(* IEC 61131-3 sources: IEC61131-3-CDSV3/Regular Expressions/src/20 Program Organization Units, 8 files *)

(* ---- FuCompiledPatternAnsiToW.pou ---- *)
(*#-#-#-#-#-#-#-#-#-#---Declaration---#-#-#-#-#-#-#-#-#-#-#-#-#*)

// Converts an ANSI/ISO 8859-1 compiled pattern to an Unicode compiled pattern.
// ANSI/ISO 8859-1 compiled patterns can be converted to Unicode without any loss.
FUNCTION FuCompiledPatternAnsiToW : typCompiledPatternW
VAR_INPUT
    typPattern: typCompiledPattern;
END_VAR
{library PRIVATE}
VAR
    i: UDINT;
END_VAR
(*#-#-#-#-#-#-#-#-#-#---Implementation---#-#-#-#-#-#-#-#-#-#-#-#-#*)

IF typPattern.uiCountTokens = 0 THEN
    RETURN;
END_IF

FuCompiledPatternAnsiToW.xCaseInsensitive := typPattern.xCaseInsensitive;
FuCompiledPatternAnsiToW.uiCountTokens := typPattern.uiCountTokens;

FOR i := 0 TO TO_UDINT((typPattern.uiCountTokens - 1)) BY 1 DO
    FuCompiledPatternAnsiToW.atTokens[i].eType := typPattern.atTokens[i].eType;
    FuCompiledPatternAnsiToW.atTokens[i].dwChar := TO_DWORD(typPattern.atTokens[i].bChar);
    FuCompiledPatternAnsiToW.atTokens[i].dwAlternativeChar := TO_DWORD(typPattern.atTokens[i].bAlternativeChar);
END_FOR

(* ---- FuCompilePattern.pou ---- *)
(*#-#-#-#-#-#-#-#-#-#---Declaration---#-#-#-#-#-#-#-#-#-#-#-#-#*)

// Compiles the pattern into a stream of tokens for matching.
// The ISO 8859-1 latin alphabet can be matched case insensitive,
// otherwise by default the pattern is case sensitive.
//
// A few examples of valid patterns:
//  - 'A*bEd'
//  - 'A*?bEd'
//  - 'A.b*e*'
//  - '*A\.b\*e*'
//  - 'A?\bed'
//
// The return value signifies whether compilation was successful,
// or the given pattern is invalid.
{attribute 'qualified_only'}
FUNCTION FuCompilePattern : BOOL
VAR_INPUT
    sPattern: STRING(255);              // The pattern string to compile
    xCaseInsensitive: BOOL := FALSE;    // Whether the pattern is case insensitive (ISO 8859-1 latin1)
END_VAR
VAR_OUTPUT
    typPattern: typCompiledPattern;     // The compiled pattern, for "FuMatchExpression"
END_VAR
{library PRIVATE}
VAR
    i: UINT;

    tempChar: BYTE;
    tempNextChar: BYTE;
    tempIndex: UINT;

    tempMaxStrIndex: UINT;
END_VAR
VAR CONSTANT
    CHAR_WILDCARD: BYTE := 42; // *
    CHAR_LAZINESS: BYTE := 63; // ?
    CHAR_DOT: BYTE := 46; // .
    CHAR_ESCAPE: BYTE := 92; // \
END_VAR
(*#-#-#-#-#-#-#-#-#-#---Implementation---#-#-#-#-#-#-#-#-#-#-#-#-#*)

FuCompilePattern := FALSE;

IF sPattern = '' THEN
    RETURN;
END_IF

tempMaxStrIndex := TO_UINT(Standard.LEN(sPattern)) - 1;

FOR i := 0 TO tempMaxStrIndex BY 1 DO
    IF sPattern[i] = 0 OR_ELSE tempIndex > ParameterList.uiMaxPatternTokens THEN
        EXIT;
    END_IF

    tempChar := TO_BYTE(sPattern[i]);

    IF i < tempMaxStrIndex THEN
        tempNextChar := TO_BYTE(sPattern[(i + 1)]);
    ELSE
        tempNextChar := 0;
    END_IF

    IF tempChar = CHAR_WILDCARD THEN // Wildcard (*)
        typPattern.atTokens[tempIndex].eType := eTokenType.WILDCARD;
        typPattern.atTokens[tempIndex].bChar := 0; // Use bChar as modifier to be lazy
    ELSIF
        tempChar = CHAR_LAZINESS AND_THEN
        tempIndex > 0 AND_THEN
        typPattern.atTokens[(tempIndex - 1)].eType = eTokenType.WILDCARD
    THEN // Laziness (?), but only if previously wildcard, otherwise literal
        typPattern.atTokens[(tempIndex - 1)].bChar := 1;
        CONTINUE;
    ELSIF tempChar = CHAR_DOT THEN // Single char (.)
        typPattern.atTokens[tempIndex].eType := eTokenType.ANYCHAR;
    ELSIF
        tempChar = CHAR_ESCAPE AND_THEN (
            tempNextChar = CHAR_WILDCARD OR_ELSE
            tempNextChar = CHAR_DOT
        )
    THEN // Backslash (escape token for . or *, if followed by . or *)
        typPattern.atTokens[tempIndex].eType := eTokenType.LITERAL;
        typPattern.atTokens[tempIndex].bChar := tempNextChar;
        i := i + 1;
    ELSE
        typPattern.atTokens[tempIndex].eType := eTokenType.LITERAL;
        typPattern.atTokens[tempIndex].bChar := tempChar;

        tempNextChar := 0;
        IF xCaseInsensitive THEN
            // Calculate for the ISO 8859-1 latin1 alphabet the uppercase or lowercase character number
            IF tempChar >= 65 AND_THEN tempChar <= 90 THEN
                // Uppercase A-Z
                tempNextChar := tempChar + 32;
            ELSIF tempChar >= 97 AND_THEN tempChar <= 122 THEN
                // Lowercase a-z
                tempNextChar := tempChar - 32;
            ELSIF tempChar >= 192 AND_THEN tempChar <= 221 AND_THEN tempChar <> 215 THEN
                // Uppercase ISO 8859-1
                tempNextChar := tempChar + 32;
            ELSIF tempChar >= 224 AND_THEN tempChar <= 253 AND_THEN tempChar <> 247 THEN
                // Lowercase ISO 8859-1
                tempNextChar := tempChar - 32;
            END_IF
        END_IF

        typPattern.atTokens[tempIndex].bAlternativeChar := tempNextChar;
    END_IF

    tempIndex := tempIndex + 1;
    typPattern.uiCountTokens := tempIndex;
END_FOR

FuCompilePattern := (tempIndex > 0);
typPattern.xCaseInsensitive := xCaseInsensitive;

(* ---- FuCompilePatternUTF8.pou ---- *)
(*#-#-#-#-#-#-#-#-#-#---Declaration---#-#-#-#-#-#-#-#-#-#-#-#-#*)

// Compiles the pattern into a stream of tokens for matching.
// This is the UTF-8 version of FuCompilePattern.
//
// Disabling strict conformity allows the usage of the extended ASCII alphabet (ISO 8859-1, decimal 160-255),
// as long as it doesn't form a valid UTF-8 byte sequence.
//
// The alphabet can be matched case insensitive,
// otherwise by default the pattern is case sensitive.
// The case mapping table is NOT completely covered,
// as such you MAY encounter missing case conversion
// for some languages.
//
// A few examples of valid patterns:
//  - 'A*bEd'
//  - 'A*?bEd'
//  - 'A.b*e*'
//  - '*A\.b\*e*'
//  - 'A?\bed'
//
// The return value signifies whether compilation was successful,
// or the given pattern is invalid.
{attribute 'qualified_only'}
FUNCTION FuCompilePatternUTF8 : BOOL
VAR_INPUT
    psPattern: POINTER TO STRING(1);      // The pattern string to compile - for technical reasons this is a STRING(1), although any length is supported
    udiPatternLength: UDINT;              // Pattern string length (in bytes, not codepoints)
    xCaseInsensitive: BOOL := FALSE;      // Whether the pattern is case insensitive
    xStrictConformity: BOOL := TRUE;      // Require strict conformity to the Unicode standard
END_VAR
VAR_OUTPUT
    typPattern: typCompiledPatternW;      // The compiled pattern, for "FuMatchExpressionUTF8"
END_VAR
{library PRIVATE}
VAR
    tempPointer: POINTER TO STRING(1);

    i: UDINT;

    tempChar: DWORD;
    tempCharLength: UDINT;

    tempNextChar: DWORD;
    tempNextCharLength: UDINT;

    tempIndex: UINT;
    tempMaxStrIndex: UDINT;
END_VAR
VAR CONSTANT
    CHAR_WILDCARD: DWORD := 42; // *
    CHAR_LAZINESS: DWORD := 63; // ?
    CHAR_DOT: DWORD := 46; // .
    CHAR_ESCAPE: DWORD := 92; // \
END_VAR
(*#-#-#-#-#-#-#-#-#-#---Implementation---#-#-#-#-#-#-#-#-#-#-#-#-#*)

FuCompilePatternUTF8 := FALSE;

IF udiPatternLength = 0 THEN
    RETURN;
END_IF

tempPointer := psPattern;

i := 0;
tempMaxStrIndex := udiPatternLength - 1;

WHILE i <= tempMaxStrIndex DO
    IF tempIndex > ParameterList.uiMaxPatternTokens THEN
        EXIT;
    END_IF

    IF
        NOT FuUtf8CharToDword(
            psInput := (tempPointer + i),
            udiStringLength := (udiPatternLength - i),
            xStrictConformity := xStrictConformity,
            dwCodepoint => tempChar,
            usiByteLength => tempCharLength
        )
    THEN
        RETURN;
    END_IF

    IF tempChar = 0 THEN
        EXIT;
    END_IF

    IF
        i > tempMaxStrIndex OR_ELSE
        NOT FuUtf8CharToDword(
            psInput := (tempPointer + i + tempCharLength),
            udiStringLength := (udiPatternLength - i),
            xStrictConformity := xStrictConformity,
            dwCodepoint => tempNextChar,
            usiByteLength => tempNextCharLength
        )
    THEN
        tempNextChar := 0;
        tempNextCharLength := 0;
    END_IF

    IF tempChar = CHAR_WILDCARD THEN // Wildcard (*)
        typPattern.atTokens[tempIndex].eType := eTokenType.WILDCARD;
        typPattern.atTokens[tempIndex].dwChar := 0; // Use dwChar as modifier to be lazy
    ELSIF
        tempChar = CHAR_LAZINESS AND_THEN
        tempIndex > 0 AND_THEN
        typPattern.atTokens[(tempIndex - 1)].eType = eTokenType.WILDCARD
    THEN // Laziness (?), but only if previously wildcard, otherwise literal
        typPattern.atTokens[(tempIndex - 1)].dwChar := 1;

        i := i + tempCharLength;
        CONTINUE;
    ELSIF tempChar = CHAR_DOT THEN // Single char (.)
        typPattern.atTokens[tempIndex].eType := eTokenType.ANYCHAR;
    ELSIF
        tempChar = CHAR_ESCAPE AND_THEN (
            tempNextChar = CHAR_WILDCARD OR_ELSE
            tempNextChar = CHAR_DOT
        )
    THEN // Backslash (escape token for . or *, if followed by . or *)
        typPattern.atTokens[tempIndex].eType := eTokenType.LITERAL;
        typPattern.atTokens[tempIndex].dwChar := tempNextChar;
        i := i + tempNextCharLength;
    ELSE
        typPattern.atTokens[tempIndex].eType := eTokenType.LITERAL;
        typPattern.atTokens[tempIndex].dwChar := tempChar;

        IF xCaseInsensitive THEN
            // Calculate for the ISO 8859-1 latin1 alphabet the uppercase or lowercase character number (efficient way)
            IF tempChar >= 65 AND_THEN tempChar <= 90 THEN
                // Uppercase A-Z
                tempNextChar := tempChar + 32;
            ELSIF tempChar >= 97 AND_THEN tempChar <= 122 THEN
                // Lowercase a-z
                tempNextChar := tempChar - 32;
            ELSIF tempChar >= 192 AND_THEN tempChar <= 221 AND_THEN tempChar <> 215 THEN
                // Uppercase ISO 8859-1
                tempNextChar := tempChar + 32;
            ELSIF tempChar >= 224 AND_THEN tempChar <= 253 AND_THEN tempChar <> 247 THEN
                // Lowercase ISO 8859-1
                tempNextChar := tempChar - 32;
            ELSE
                // If we're not in the ISO 8859-1 latin1 alphabet range, use the Unicode function to calculate it
                tempNextChar := FuUnicodeCodepointCaseConvert(tempChar);
            END_IF
        ELSE
            tempNextChar := 0;
        END_IF

        typPattern.atTokens[tempIndex].dwAlternativeChar := tempNextChar;
    END_IF

    tempIndex := tempIndex + 1;
    typPattern.uiCountTokens := tempIndex;

    i := i + tempCharLength;
END_WHILE

FuCompilePatternUTF8 := (tempIndex > 0);
typPattern.xCaseInsensitive := xCaseInsensitive;

(* ---- FuCompilePatternW.pou ---- *)
(*#-#-#-#-#-#-#-#-#-#---Declaration---#-#-#-#-#-#-#-#-#-#-#-#-#*)

// Compiles the pattern into a stream of tokens for matching.
// This is the UTF-16 (WSTRING) version of FuCompilePattern.
//
// The alphabet can be matched case insensitive,
// otherwise by default the pattern is case sensitive.
// The case mapping table is NOT completely covered,
// as such you MAY encounter missing case conversion
// for some languages.
//
// A few examples of valid patterns:
//  - 'A*bEd'
//  - 'A*?bEd'
//  - 'A.b*e*'
//  - '*A\.b\*e*'
//  - 'A?\bed'
//
// The return value signifies whether compilation was successful,
// or the given pattern is invalid.
{attribute 'qualified_only'}
FUNCTION FuCompilePatternW : BOOL
VAR_INPUT
    pwsPattern: POINTER TO WSTRING(1);    // The pattern string to compile - for technical reasons this is a WSTRING(1), although any length is supported
    udiPatternLength: UDINT;              // Pattern string length (in words (length in bytes/2), not codepoints)
    xCaseInsensitive: BOOL := FALSE;      // Whether the pattern is case insensitive
END_VAR
VAR_OUTPUT
    typPattern: typCompiledPatternW;      // The compiled pattern, for "FuMatchExpressionW"
END_VAR
{library PRIVATE}
VAR
    tempPointer: POINTER TO WSTRING(1);

    i: UDINT;

    tempChar: DWORD;
    tempCharLength: UDINT;

    tempNextChar: DWORD;
    tempNextCharLength: UDINT;

    tempIndex: UINT;
    tempMaxStrIndex: UDINT;
END_VAR
VAR CONSTANT
    CHAR_WILDCARD: DWORD := 42; // *
    CHAR_LAZINESS: DWORD := 63; // ?
    CHAR_DOT: DWORD := 46; // .
    CHAR_ESCAPE: DWORD := 92; // \
END_VAR
(*#-#-#-#-#-#-#-#-#-#---Implementation---#-#-#-#-#-#-#-#-#-#-#-#-#*)

FuCompilePatternW := FALSE;

IF udiPatternLength = 0 THEN
    RETURN;
END_IF

tempPointer := pwsPattern;

i := 0;
tempMaxStrIndex := udiPatternLength - 1;

WHILE i <= tempMaxStrIndex DO
    IF tempIndex > ParameterList.uiMaxPatternTokens THEN
        EXIT;
    END_IF

    IF NOT FuUtf16CharToDword(psInput := (tempPointer + (i * 2)), udiStringLength := (udiPatternLength - (i * 2)), dwCodepoint => tempChar, usiWordLength => tempCharLength) THEN
        RETURN;
    END_IF

    IF tempChar = 0 THEN
        EXIT;
    END_IF

    IF
        i > tempMaxStrIndex OR_ELSE
        NOT FuUtf16CharToDword(
            psInput := (tempPointer + (i * 2) + (tempCharLength * 2)),
            udiStringLength := (udiPatternLength - (i * 2) - (tempCharLength * 2)),
            dwCodepoint => tempNextChar,
            usiWordLength => tempNextCharLength
        )
    THEN
        tempNextChar := 0;
        tempNextCharLength := 0;
    END_IF

    IF tempChar = CHAR_WILDCARD THEN // Wildcard (*)
        typPattern.atTokens[tempIndex].eType := eTokenType.WILDCARD;
        typPattern.atTokens[tempIndex].dwChar := 0; // Use dwChar as modifier to be lazy
    ELSIF
        tempChar = CHAR_LAZINESS AND_THEN
        tempIndex > 0 AND_THEN
        typPattern.atTokens[(tempIndex - 1)].eType = eTokenType.WILDCARD
    THEN // Laziness (?), but only if previously wildcard, otherwise literal
        typPattern.atTokens[(tempIndex - 1)].dwChar := 1;

        i := i + tempCharLength;
        CONTINUE;
    ELSIF tempChar = CHAR_DOT THEN // Single char (.)
        typPattern.atTokens[tempIndex].eType := eTokenType.ANYCHAR;
    ELSIF
        tempChar = CHAR_ESCAPE AND_THEN (
            tempNextChar = CHAR_WILDCARD OR_ELSE
            tempNextChar = CHAR_DOT
        )
    THEN // Backslash (escape token for . or *, if followed by . or *)
        typPattern.atTokens[tempIndex].eType := eTokenType.LITERAL;
        typPattern.atTokens[tempIndex].dwChar := tempNextChar;
        i := i + tempNextCharLength;
    ELSE
        typPattern.atTokens[tempIndex].eType := eTokenType.LITERAL;
        typPattern.atTokens[tempIndex].dwChar := tempChar;

        IF xCaseInsensitive THEN
            // Calculate for the ISO 8859-1 latin1 alphabet the uppercase or lowercase character number (efficient way)
            IF tempChar >= 65 AND_THEN tempChar <= 90 THEN
                // Uppercase A-Z
                tempNextChar := tempChar + 32;
            ELSIF tempChar >= 97 AND_THEN tempChar <= 122 THEN
                // Lowercase a-z
                tempNextChar := tempChar - 32;
            ELSIF tempChar >= 192 AND_THEN tempChar <= 221 AND_THEN tempChar <> 215 THEN
                // Uppercase ISO 8859-1
                tempNextChar := tempChar + 32;
            ELSIF tempChar >= 224 AND_THEN tempChar <= 253 AND_THEN tempChar <> 247 THEN
                // Lowercase ISO 8859-1
                tempNextChar := tempChar - 32;
            ELSE
                // If we're not in the ISO 8859-1 latin1 alphabet range, use the UTF-8 function to calculate it
                tempNextChar := FuUnicodeCodepointCaseConvert(tempChar);
            END_IF
        ELSE
            tempNextChar := 0;
        END_IF

        typPattern.atTokens[tempIndex].dwAlternativeChar := tempNextChar;
    END_IF

    tempIndex := tempIndex + 1;
    typPattern.uiCountTokens := tempIndex;

    i := i + tempCharLength;
END_WHILE

FuCompilePatternW := (tempIndex > 0);
typPattern.xCaseInsensitive := xCaseInsensitive;

(* ---- FuCompilePatternW2.pou ---- *)
(*#-#-#-#-#-#-#-#-#-#---Declaration---#-#-#-#-#-#-#-#-#-#-#-#-#*)

// Same as FuCompilePatternW, except it doesn't take a pointer and has a fixed length.
{attribute 'qualified_only'}
FUNCTION FuCompilePatternW2 : BOOL
VAR_INPUT
    wsPattern: WSTRING(255);              // The pattern string to compile
    xCaseInsensitive: BOOL := FALSE;      // Whether the pattern is case insensitive
END_VAR
VAR_OUTPUT
    typPattern: typCompiledPatternW;      // The compiled pattern, for "FuMatchExpressionW"
END_VAR
(*#-#-#-#-#-#-#-#-#-#---Implementation---#-#-#-#-#-#-#-#-#-#-#-#-#*)

FuCompilePatternW2 := FuCompilePatternW(ADR(wsPattern), TO_UDINT(Stu.StrLenW(ADR(wsPattern))), xCaseInsensitive, typPattern => typPattern);

(* ---- FuMatchExpression.pou ---- *)
(*#-#-#-#-#-#-#-#-#-#---Declaration---#-#-#-#-#-#-#-#-#-#-#-#-#*)

// Matches the given compiled pattern against the subject.
{attribute 'qualified_only'}
FUNCTION FuMatchExpression : BOOL
VAR_INPUT
    typPattern: typCompiledPattern;     // The compiled pattern from "FuCompilePattern"
    psSubject: POINTER TO STRING(1);    // A pointer to the subject string - for technical reasons this is a STRING(1), although any size is supported
    udiLength: UDINT;                   // The length of the subject string
END_VAR
{library PRIVATE}
VAR
    tempPtrStr: POINTER TO BYTE;
    tempPtrStrMatching: POINTER TO BYTE;
    tempStrIndex: UDINT;
    tempStrIndexMatching: UDINT;

    i: UINT;
    j: UINT;
    k: LINT;

    tempLaziness: BOOL;
    tempHasEndChar: BOOL;
    tempEndChar: BYTE;
    tempEndChar2: BYTE;

    tempWildcardSearchStart: LINT;
    tempWildcardSearchEnd: LINT;
    tempWildcardSearchBy: LINT;
    tempWildcardSearchSuccess: BOOL;
END_VAR
(*#-#-#-#-#-#-#-#-#-#---Implementation---#-#-#-#-#-#-#-#-#-#-#-#-#*)

FuMatchExpression := FALSE;

IF typPattern.uiCountTokens = 0 OR_ELSE udiLength = 0 THEN
    RETURN;
END_IF

tempPtrStr := psSubject;
tempStrIndex := 0;

WHILE i < typPattern.uiCountTokens DO
    IF tempStrIndex >= udiLength THEN
        // Only if all following tokens are of type WILDCARD, we can allow a match to be positive
        FOR j := i TO (typPattern.uiCountTokens - 1) BY 1 DO
            IF typPattern.atTokens[j].eType <> eTokenType.WILDCARD THEN
                FuMatchExpression := FALSE;
                RETURN;
            END_IF
        END_FOR

        FuMatchExpression := TRUE;
        RETURN;
    END_IF

    CASE typPattern.atTokens[i].eType OF
        eTokenType.INVALID: // We shouldn't ever get an invalid token inside our token array that isn't behind our count
            RETURN;

        eTokenType.LITERAL:
            IF
                tempPtrStr[tempStrIndex] <> typPattern.atTokens[i].bChar AND_THEN
                (
                    NOT typPattern.xCaseInsensitive OR_ELSE (
                        typPattern.atTokens[i].bAlternativeChar <> 0 AND_THEN
                        tempPtrStr[tempStrIndex] <> typPattern.atTokens[i].bAlternativeChar
                    )
                )
            THEN
                RETURN;
            END_IF

            tempStrIndex := tempStrIndex + 1;

        eTokenType.ANYCHAR:
            tempStrIndex := tempStrIndex + 1;

        eTokenType.WILDCARD:
            tempLaziness := (typPattern.atTokens[i].bChar = 1);
            tempHasEndChar := FALSE;

            FOR j := i + 1 TO (typPattern.uiCountTokens - 1) BY 1 DO
                IF typPattern.atTokens[j].eType = eTokenType.LITERAL THEN
                    tempHasEndChar := TRUE;
                    tempEndChar := typPattern.atTokens[j].bChar;
                    tempEndChar2 := typPattern.atTokens[j].bAlternativeChar;
                    EXIT;
                END_IF
            END_FOR

            // If we don't have any characters to match on at the end of the pattern, we match immediately
            IF NOT tempHasEndChar THEN
                FuMatchExpression := TRUE;
                RETURN;
            END_IF

            IF tempLaziness THEN
                // Advance token pointer once more because the next token is the laziness token we already used
                i := i + 1;

                // If the wildcard is lazy, search from front to back
                tempWildcardSearchStart := TO_LINT(tempStrIndex);
                tempWildcardSearchEnd := TO_LINT(udiLength);
                tempWildcardSearchBy := 1;
            ELSE
                // If the wildcard is NOT lazy, search from back to front (greedy!)
                tempWildcardSearchStart := TO_LINT(udiLength);
                tempWildcardSearchEnd := TO_LINT(tempStrIndex);
                tempWildcardSearchBy := -1;
            END_IF

            tempWildcardSearchSuccess := FALSE;
            FOR k := tempWildcardSearchStart TO tempWildcardSearchEnd BY tempWildcardSearchBy DO
                IF
                    tempPtrStr[k] = tempEndChar OR_ELSE
                    (typPattern.xCaseInsensitive AND_THEN tempEndChar2 <> 0 AND_THEN tempPtrStr[k] = tempEndChar2)
                THEN
                    tempWildcardSearchSuccess := TRUE;
                    tempStrIndex := TO_UDINT(k);
                    EXIT;
                END_IF
            END_FOR

            IF NOT tempWildcardSearchSuccess THEN
                RETURN;
            END_IF
    END_CASE

    i := i + 1;
END_WHILE

FuMatchExpression := (tempStrIndex >= udiLength);

(* ---- FuMatchExpressionUTF8.pou ---- *)
(*#-#-#-#-#-#-#-#-#-#---Declaration---#-#-#-#-#-#-#-#-#-#-#-#-#*)

// Matches the given compiled pattern against the subject.
// This is the UTF-8 version of FuMatchExpression.
// Disabling strict conformity allows the usage of the extended ASCII alphabet (ISO 8859-1, decimal 160-255),
// as long as it doesn't form a valid UTF-8 byte sequence.
{attribute 'qualified_only'}
FUNCTION FuMatchExpressionUTF8 : BOOL
VAR_INPUT
    typPattern: typCompiledPatternW;      // The compiled pattern from "FuCompilePatternW"
    psSubject: POINTER TO STRING(1);      // A pointer to the subject string - for technical reasons this is a STRING(1), although any size is supported
    udiLength: UDINT;                     // The length of the subject string (in bytes, not codepoints)
    xStrictConformity: BOOL := TRUE;      // Require strict conformity to the Unicode standard
END_VAR
{library PRIVATE}
VAR
    tempPtrStr: POINTER TO BYTE;
    tempPtrStrMatching: POINTER TO BYTE;
    tempStrIndex: UDINT;
    tempStrIndexMatching: UDINT;

    i: UINT;
    j: UINT;
    k: LINT;

    tempChar: DWORD;
    tempCharLength: USINT;

    tempNextChar: DWORD;
    tempNextCharLength: DWORD;

    tempLaziness: BOOL;
    tempHasEndChar: BOOL;
    tempEndChar: DWORD;
    tempEndChar2: DWORD;

    tempWildcardSearchStart: LINT;
    tempWildcardSearchEnd: LINT;
    tempWildcardSearchBy: LINT;
    tempWildcardSearchOffset: UDINT;
    tempWildcardSearchSuccess: BOOL;
END_VAR
(*#-#-#-#-#-#-#-#-#-#---Implementation---#-#-#-#-#-#-#-#-#-#-#-#-#*)

FuMatchExpressionUTF8 := FALSE;

IF typPattern.uiCountTokens = 0 OR_ELSE udiLength = 0 THEN
    RETURN;
END_IF

tempPtrStr := psSubject;
tempStrIndex := 0;

WHILE i < typPattern.uiCountTokens DO
    IF tempStrIndex >= udiLength THEN
        // Only if all following tokens are of type WILDCARD, we can allow a match to be positive
        FOR j := i TO (typPattern.uiCountTokens - 1) BY 1 DO
            IF typPattern.atTokens[j].eType <> eTokenType.WILDCARD THEN
                FuMatchExpressionUTF8 := FALSE;
                RETURN;
            END_IF
        END_FOR

        FuMatchExpressionUTF8 := TRUE;
        RETURN;
    END_IF

    IF
        NOT FuUtf8CharToDword(
            psInput := (tempPtrStr + tempStrIndex),
            udiStringLength := (udiLength - tempStrIndex),
            xStrictConformity := xStrictConformity,
            dwCodepoint => tempChar,
            usiByteLength => tempCharLength
        )
    THEN
        RETURN;
    END_IF

    CASE typPattern.atTokens[i].eType OF
        eTokenType.INVALID: // We shouldn't ever get an invalid token inside our token array that isn't behind our count
            RETURN;

        eTokenType.LITERAL:
            IF
                tempChar <> typPattern.atTokens[i].dwChar AND_THEN
                (
                    NOT typPattern.xCaseInsensitive OR_ELSE
                    typPattern.atTokens[i].dwAlternativeChar = 0 OR_ELSE
                    tempChar <> typPattern.atTokens[i].dwAlternativeChar
                )
            THEN
                RETURN;
            END_IF

            tempStrIndex := tempStrIndex + tempCharLength;

        eTokenType.ANYCHAR:
            tempStrIndex := tempStrIndex + tempCharLength;

        eTokenType.WILDCARD:
            tempLaziness := (typPattern.atTokens[i].dwChar = 1);
            tempHasEndChar := FALSE;

            FOR j := i + 1 TO (typPattern.uiCountTokens - 1) BY 1 DO
                IF typPattern.atTokens[j].eType = eTokenType.LITERAL THEN
                    tempHasEndChar := TRUE;
                    tempEndChar := typPattern.atTokens[j].dwChar;
                    tempEndChar2 := typPattern.atTokens[j].dwAlternativeChar;
                    EXIT;
                END_IF
            END_FOR

            // If we don't have any characters to match on at the end of the pattern, we match immediately
            IF NOT tempHasEndChar THEN
                FuMatchExpressionUTF8 := TRUE;
                RETURN;
            END_IF

            IF tempLaziness THEN
                // Advance token pointer once more because the next token is the laziness token we already used
                i := i + 1;

                // If the wildcard is lazy, search from front to back
                tempWildcardSearchStart := TO_LINT(tempStrIndex);
                tempWildcardSearchEnd := TO_LINT(udiLength);
                tempWildcardSearchBy := 1;
            ELSE
                // If the wildcard is NOT lazy, search from back to front (greedy!)
                tempWildcardSearchStart := TO_LINT(udiLength);
                tempWildcardSearchEnd := TO_LINT(tempStrIndex);
                tempWildcardSearchBy := -1;
            END_IF

            tempWildcardSearchSuccess := FALSE;
            tempWildcardSearchOffset := 0;

            FOR k := tempWildcardSearchStart TO tempWildcardSearchEnd BY tempWildcardSearchBy DO
                IF
                    FuUtf8CharToDword(
                        psInput := (tempPtrStr + LINT_TO___XWORD(k)),
                        udiStringLength := (udiLength - tempWildcardSearchOffset),
                        xStrictConformity := xStrictConformity,
                        dwCodepoint => tempNextChar,
                        usiByteLength => tempNextCharLength
                    )
                THEN
                    tempWildcardSearchOffset := tempWildcardSearchOffset + tempNextCharLength;

                    IF
                        tempNextChar = tempEndChar OR_ELSE
                        (typPattern.xCaseInsensitive AND_THEN tempEndChar2 <> 0 AND_THEN tempNextChar = tempEndChar2)
                    THEN
                        tempWildcardSearchSuccess := TRUE;
                        tempStrIndex := TO_UDINT(k);
                        EXIT;
                    END_IF
                ELSE
                    tempWildcardSearchOffset := tempWildcardSearchOffset + 1;
                END_IF
            END_FOR

            IF NOT tempWildcardSearchSuccess THEN
                RETURN;
            END_IF
    END_CASE

    i := i + 1;
END_WHILE

FuMatchExpressionUTF8 := (tempStrIndex >= udiLength);

(* ---- FuMatchExpressionW.pou ---- *)
(*#-#-#-#-#-#-#-#-#-#---Declaration---#-#-#-#-#-#-#-#-#-#-#-#-#*)

// Matches the given compiled pattern against the subject.
// This is the UTF-16 (WSTRING) version of FuMatchExpression.
{attribute 'qualified_only'}
FUNCTION FuMatchExpressionW : BOOL
VAR_INPUT
    typPattern: typCompiledPatternW;      // The compiled pattern from "FuCompilePatternW"
    pwsSubject: POINTER TO WSTRING(1);    // A pointer to the subject string - for technical reasons this is a WSTRING(1), although any size is supported
    udiLength: UDINT;                     // The length of the subject string (in words (length in bytes/2), not codepoints)
END_VAR
{library PRIVATE}
VAR
    tempPtrStr: POINTER TO WORD;
    tempPtrStrMatching: POINTER TO WORD;
    tempStrIndex: UDINT;
    tempStrIndexMatching: UDINT;

    i: UINT;
    j: UINT;
    k: LINT;

    tempChar: DWORD;
    tempCharLength: USINT;

    tempNextChar: DWORD;
    tempNextCharLength: DWORD;

    tempLaziness: BOOL;
    tempHasEndChar: BOOL;
    tempEndChar: DWORD;
    tempEndChar2: DWORD;

    tempWildcardSearchStart: LINT;
    tempWildcardSearchEnd: LINT;
    tempWildcardSearchBy: LINT;
    tempWildcardSearchOffset: UDINT;
    tempWildcardSearchSuccess: BOOL;
END_VAR
(*#-#-#-#-#-#-#-#-#-#---Implementation---#-#-#-#-#-#-#-#-#-#-#-#-#*)

FuMatchExpressionW := FALSE;

IF typPattern.uiCountTokens = 0 OR_ELSE udiLength = 0 THEN
    RETURN;
END_IF

tempPtrStr := pwsSubject;
tempStrIndex := 0;

WHILE i < typPattern.uiCountTokens DO
    IF tempStrIndex >= udiLength THEN
        // Only if all following tokens are of type WILDCARD, we can allow a match to be positive
        FOR j := i TO (typPattern.uiCountTokens - 1) BY 1 DO
            IF typPattern.atTokens[j].eType <> eTokenType.WILDCARD THEN
                FuMatchExpressionW := FALSE;
                RETURN;
            END_IF
        END_FOR

        FuMatchExpressionW := TRUE;
        RETURN;
    END_IF

    IF NOT FuUtf16CharToDword(psInput := (tempPtrStr + (tempStrIndex * 2)), udiStringLength := (udiLength - (tempStrIndex * 2)), dwCodepoint => tempChar, usiWordLength => tempCharLength) THEN
        RETURN;
    END_IF

    CASE typPattern.atTokens[i].eType OF
        eTokenType.INVALID: // We shouldn't ever get an invalid token inside our token array that isn't behind our count
            RETURN;

        eTokenType.LITERAL:
            IF
                tempChar <> typPattern.atTokens[i].dwChar AND_THEN
                (
                    NOT typPattern.xCaseInsensitive OR_ELSE
                    typPattern.atTokens[i].dwAlternativeChar = 0 OR_ELSE
                    tempChar <> typPattern.atTokens[i].dwAlternativeChar
                )
            THEN
                RETURN;
            END_IF

            tempStrIndex := tempStrIndex + tempCharLength;

        eTokenType.ANYCHAR:
            tempStrIndex := tempStrIndex + tempCharLength;

        eTokenType.WILDCARD:
            tempLaziness := (typPattern.atTokens[i].dwChar = 1);
            tempHasEndChar := FALSE;

            FOR j := i + 1 TO (typPattern.uiCountTokens - 1) BY 1 DO
                IF typPattern.atTokens[j].eType = eTokenType.LITERAL THEN
                    tempHasEndChar := TRUE;
                    tempEndChar := typPattern.atTokens[j].dwChar;
                    tempEndChar2 := typPattern.atTokens[j].dwAlternativeChar;
                    EXIT;
                END_IF
            END_FOR

            // If we don't have any characters to match on at the end of the pattern, we match immediately
            IF NOT tempHasEndChar THEN
                FuMatchExpressionW := TRUE;
                RETURN;
            END_IF

            IF tempLaziness THEN
                // Advance token pointer once more because the next token is the laziness token we already used
                i := i + 1;

                // If the wildcard is lazy, search from front to back
                tempWildcardSearchStart := TO_LINT(tempStrIndex);
                tempWildcardSearchEnd := TO_LINT(udiLength);
                tempWildcardSearchBy := 1;
            ELSE
                // If the wildcard is NOT lazy, search from back to front (greedy!)
                tempWildcardSearchStart := TO_LINT(udiLength);
                tempWildcardSearchEnd := TO_LINT(tempStrIndex);
                tempWildcardSearchBy := -1;
            END_IF

            tempWildcardSearchSuccess := FALSE;
            tempWildcardSearchOffset := 0;

            FOR k := tempWildcardSearchStart TO tempWildcardSearchEnd BY tempWildcardSearchBy DO
                IF
                    FuUtf16CharToDword(
                        psInput := (tempPtrStr + LINT_TO___XWORD(k)),
                        udiStringLength := (udiLength - tempWildcardSearchOffset),
                        dwCodepoint => tempNextChar,
                        usiWordLength => tempNextCharLength
                    )
                THEN
                    tempWildcardSearchOffset := tempWildcardSearchOffset + tempNextCharLength;

                    IF
                        tempNextChar = tempEndChar OR_ELSE
                        (typPattern.xCaseInsensitive AND_THEN tempEndChar2 <> 0 AND_THEN tempNextChar = tempEndChar2)
                    THEN
                        tempWildcardSearchSuccess := TRUE;
                        tempStrIndex := TO_UDINT(k);
                        EXIT;
                    END_IF
                ELSE
                    tempWildcardSearchOffset := tempWildcardSearchOffset + 1;
                END_IF
            END_FOR

            IF NOT tempWildcardSearchSuccess THEN
                RETURN;
            END_IF
    END_CASE

    i := i + 1;
END_WHILE

FuMatchExpressionW := (tempStrIndex >= udiLength);
